Staubli VAL3: CreatFile.pgx

public program CreatFile(string x_sFileName (dimensions=1), bool& x_bRes (dimensions=1))
begin

  x_bRes=false
  nFileID=$fileOpen(x_sFileName,"w")
  if nFileID<0 or nFileID>9
    return
  endIf
  x_bRes=true
  call CloseAllFile()


end
